// TIA Portal V20 export
FUNCTION_BLOCK "MotorSequenceGRAPH"   // FB2, GRAPH
// stored: AutoNumber false, GraphVersion 6.0, SetENOAutomatically false
   // inherited from GRAPH_BASE
   VAR_INPUT
      OFF_SQ { ExternalAccessible := 'False'; ExternalVisible := 'False'; ExternalWritable := 'False'} : Bool := false;   // 关闭顺控器
      INIT_SQ { ExternalAccessible := 'False'; ExternalVisible := 'False'; ExternalWritable := 'False'} : Bool := false;   // 将顺序设置为初始状态
      ACK_EF { ExternalAccessible := 'False'; ExternalVisible := 'False'; ExternalWritable := 'False'} : Bool := false;   // 确认所有的错误和故障
      S_PREV { ExternalAccessible := 'False'; ExternalVisible := 'False'; ExternalWritable := 'False'} : Bool := false;   // 在S_NO输出参数中显示前导步
      S_NEXT { ExternalAccessible := 'False'; ExternalVisible := 'False'; ExternalWritable := 'False'} : Bool := false;   // 在S_NO输出参数中显示后续步。
      SW_AUTO { ExternalAccessible := 'False'; ExternalVisible := 'False'; ExternalWritable := 'False'} : Bool := false;   // 自动模式
      SW_TAP { ExternalAccessible := 'False'; ExternalVisible := 'False'; ExternalWritable := 'False'} : Bool := false;   // 半自动/转换条件切换
      SW_TOP { ExternalAccessible := 'False'; ExternalVisible := 'False'; ExternalWritable := 'False'} : Bool := false;   // 半自动/忽略转换条件
      SW_MAN { ExternalAccessible := 'False'; ExternalVisible := 'False'; ExternalWritable := 'False'} : Bool := false;   // 手动模式
      S_SEL { ExternalAccessible := 'False'; ExternalVisible := 'False'; ExternalWritable := 'False'} : Int := 0;   // 选择要在 S_NO中输出的步。
      S_ON { ExternalAccessible := 'False'; ExternalVisible := 'False'; ExternalWritable := 'False'} : Bool := false;   // 激活S_NO 中显示的步。
      S_OFF { ExternalAccessible := 'False'; ExternalVisible := 'False'; ExternalWritable := 'False'} : Bool := false;   // 禁用 S_NO 中标识的步
      T_PUSH { ExternalAccessible := 'False'; ExternalVisible := 'False'; ExternalWritable := 'False'} : Bool := false;   // 允许在半自动模式下跳过转换条件。
   END_VAR
   VAR_OUTPUT
      S_NO { ExternalAccessible := 'False'; ExternalVisible := 'False'; ExternalWritable := 'False'} : Int := 0;   // 步编号
      S_MORE { ExternalAccessible := 'False'; ExternalVisible := 'False'; ExternalWritable := 'False'} : Bool := false;   // 更多步可用，并可在S_NO中显示。
      S_ACTIVE { ExternalAccessible := 'False'; ExternalVisible := 'False'; ExternalWritable := 'False'} : Bool := false;   // 在S_NO 中显示的步是激活的。
      ERR_FLT { ExternalAccessible := 'False'; ExternalVisible := 'False'; ExternalWritable := 'False'} : Bool := false;   // 互锁条件或监控条件组出错
      AUTO_ON { ExternalAccessible := 'False'; ExternalVisible := 'False'; ExternalWritable := 'False'} : Bool := false;   // 当前为自动模式
      TAP_ON { ExternalAccessible := 'False'; ExternalVisible := 'False'; ExternalWritable := 'False'} : Bool := false;   // 已启用SW_TAP模式。
      TOP_ON { ExternalAccessible := 'False'; ExternalVisible := 'False'; ExternalWritable := 'False'} : Bool := false;   // 启用半自动模式/忽略转换条件。
      MAN_ON { ExternalAccessible := 'False'; ExternalVisible := 'False'; ExternalWritable := 'False'} : Bool := false;   // 已启用手动模式。
   END_VAR
BEGIN
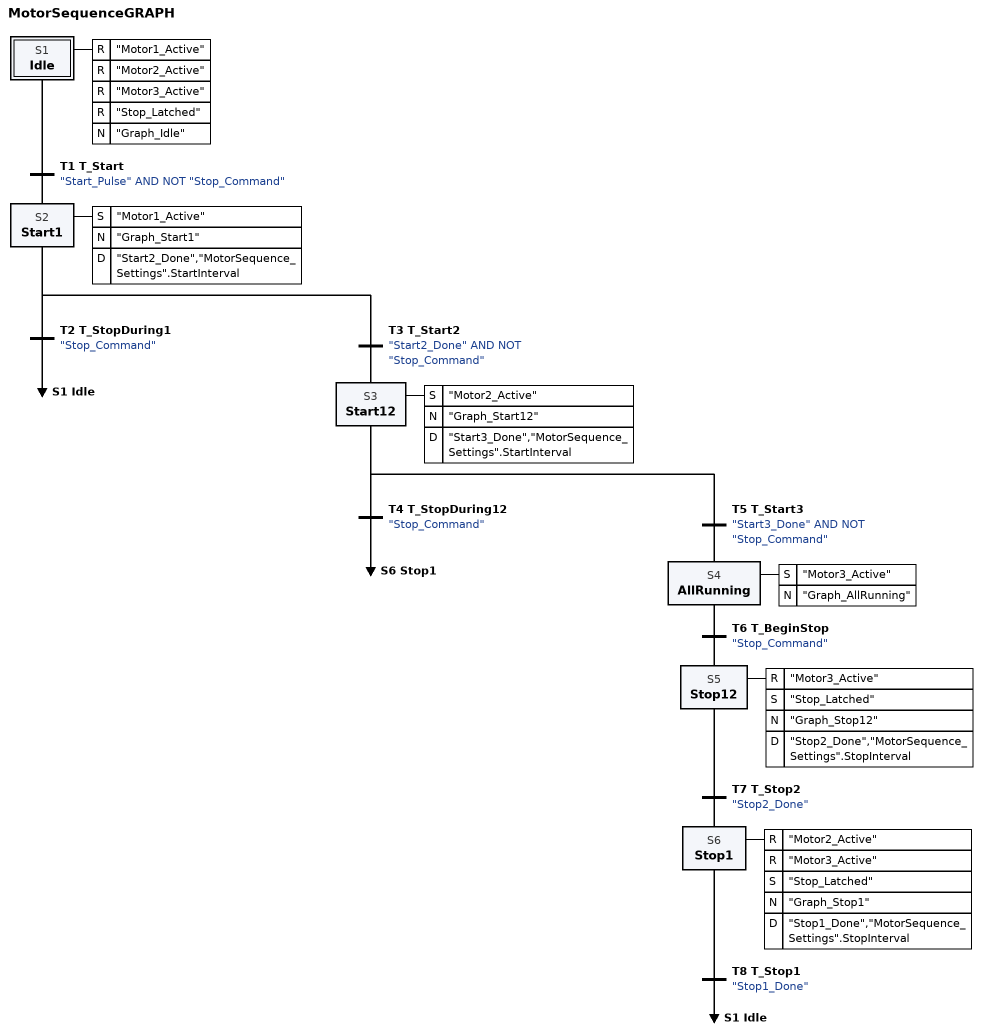
   // permanent pre-instructions
   NETWORK 1
      "Start_Pulse" := "Start_Command" AND NOT "Start_Previous";

   // sequencer 1: 三电机顺序启停：DB2可设间隔
   // 停止优先；停止阶段保持到全部停止；长按启动不自动重启。使用GRAPH原生D延时动作。
   INITIAL_STEP Idle:   // S1, max time T#0ms, warning time T#0ms
      supervision V := "Stop_Command" AND NOT "Stop_Command";
      // 空闲：全部停止，等待新的启动上升沿
              R    "Motor1_Active"
              R    "Motor2_Active"
              R    "Motor3_Active"
              R    "Stop_Latched"
              N    "Graph_Idle"
   END_STEP
   TRANSITION T_Start FROM Idle TO Start1   // T1
      := "Start_Pulse" AND NOT "Stop_Command";
   END_TRANSITION
   STEP Start1:   // S2, max time T#0ms, warning time T#0ms
      supervision V := "Stop_Command" AND NOT "Stop_Command";
      // 1号运行：等待启动间隔，停止优先
              S    "Motor1_Active"
              N    "Graph_Start1"
              D    "Start2_Done","MotorSequence_Settings".StartInterval
   END_STEP
   TRANSITION T_StopDuring1 FROM Start1 TO Idle   // T2, jump
      := "Stop_Command";
   END_TRANSITION
   TRANSITION T_Start2 FROM Start1 TO Start12   // T3
      := "Start2_Done" AND NOT "Stop_Command";
   END_TRANSITION
   STEP Start12:   // S3, max time T#0ms, warning time T#0ms
      supervision V := "Stop_Command" AND NOT "Stop_Command";
      // 1、2号运行：等待启动间隔，停止可跳至只留1号
              S    "Motor2_Active"
              N    "Graph_Start12"
              D    "Start3_Done","MotorSequence_Settings".StartInterval
   END_STEP
   TRANSITION T_StopDuring12 FROM Start12 TO Stop1   // T4, jump
      := "Stop_Command";
   END_TRANSITION
   TRANSITION T_Start3 FROM Start12 TO AllRunning   // T5
      := "Start3_Done" AND NOT "Stop_Command";
   END_TRANSITION
   STEP AllRunning:   // S4, max time T#0ms, warning time T#0ms
      supervision V := "Stop_Command" AND NOT "Stop_Command";
      // 三台电机全部运行，等待停止
              S    "Motor3_Active"
              N    "Graph_AllRunning"
   END_STEP
   TRANSITION T_BeginStop FROM AllRunning TO Stop12   // T6
      := "Stop_Command";
   END_TRANSITION
   STEP Stop12:   // S5, max time T#0ms, warning time T#0ms
      supervision V := "Stop_Command" AND NOT "Stop_Command";
      // 立即停3号，锁存停止序列，等待停止间隔
              R    "Motor3_Active"
              S    "Stop_Latched"
              N    "Graph_Stop12"
              D    "Stop2_Done","MotorSequence_Settings".StopInterval
   END_STEP
   TRANSITION T_Stop2 FROM Stop12 TO Stop1   // T7
      := "Stop2_Done";
   END_TRANSITION
   STEP Stop1:   // S6, max time T#0ms, warning time T#0ms
      supervision V := "Stop_Command" AND NOT "Stop_Command";
      // 立即停2号，保持1号至停止间隔结束
              R    "Motor2_Active"
              R    "Motor3_Active"
              S    "Stop_Latched"
              N    "Graph_Stop1"
              D    "Stop1_Done","MotorSequence_Settings".StopInterval
   END_STEP
   TRANSITION T_Stop1 FROM Stop1 TO Idle   // T8, jump
      := "Stop1_Done";
   END_TRANSITION

   // permanent post-instructions
   NETWORK 1
      "Motor_1" := "Motor1_Active";
   NETWORK 2
      "Motor_2" := "Motor2_Active";
   NETWORK 3
      "Motor_3" := "Motor3_Active";
   NETWORK 4
      "Start_Previous" := "Start_Command";
END_FUNCTION_BLOCK
